SUBAPPLICATION Uebung_049 (* DigitalInput_I1-_I4 auf DigitalOutput_Q1-_Q4 *)
  (* Standard: 61499-2; Description: Copyright (c) 2023 Meisterschulen am Ostbahnhof This program and the accompanying materials are made available under the terms of the Eclipse Public License 2.0 which is available at https://www.eclipse.org/legal/epl-2.0/ SPDX-License-Identifier: EPL-2.0 *)
  (* Version 1.0, 2023-10-23, Franz Höpfinger, Meisterschulen am Ostbahnhof *)
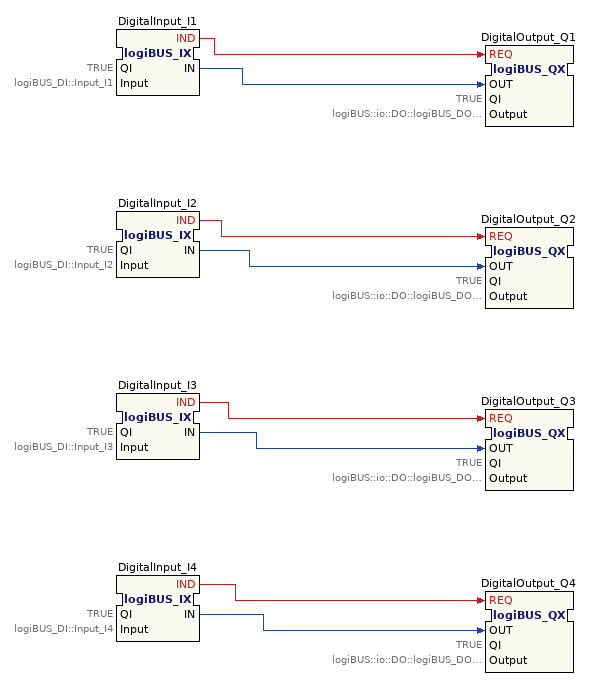
  FBS
    DigitalOutput_Q1 : logiBUS_QX(QI := TRUE, Output := logiBUS::io::DO::logiBUS_DO::Output_Q1);
    DigitalInput_I1 : logiBUS_IX(QI := TRUE, Input := logiBUS_DI::Input_I1);
    DigitalOutput_Q2 : logiBUS_QX(QI := TRUE, Output := logiBUS::io::DO::logiBUS_DO::Output_Q2);
    DigitalInput_I2 : logiBUS_IX(QI := TRUE, Input := logiBUS_DI::Input_I2);
    DigitalOutput_Q3 : logiBUS_QX(QI := TRUE, Output := logiBUS::io::DO::logiBUS_DO::Output_Q3);
    DigitalInput_I3 : logiBUS_IX(QI := TRUE, Input := logiBUS_DI::Input_I3);
    DigitalOutput_Q4 : logiBUS_QX(QI := TRUE, Output := logiBUS::io::DO::logiBUS_DO::Output_Q4);
    DigitalInput_I4 : logiBUS_IX(QI := TRUE, Input := logiBUS_DI::Input_I4);
  END_FBS
  EVENT_CONNECTIONS
    DigitalInput_I1.IND TO DigitalOutput_Q1.REQ;
    DigitalInput_I2.IND TO DigitalOutput_Q2.REQ;
    DigitalInput_I3.IND TO DigitalOutput_Q3.REQ;
    DigitalInput_I4.IND TO DigitalOutput_Q4.REQ;
  END_CONNECTIONS
  DATA_CONNECTIONS
    DigitalInput_I1.IN TO DigitalOutput_Q1.OUT;
    DigitalInput_I2.IN TO DigitalOutput_Q2.OUT;
    DigitalInput_I3.IN TO DigitalOutput_Q3.OUT;
    DigitalInput_I4.IN TO DigitalOutput_Q4.OUT;
  END_CONNECTIONS
END_SUBAPPLICATION
